PROGRAM DNS_DYN_DEMO
VAR
	DNS_DYN : DNS_DYN;
	IP_C : IP_C;
	S_BUF : NETWORK_BUFFER;
	R_BUF : NETWORK_BUFFER;
	IP_CONTROL : IP_CONTROL;
	enable: BOOL;
	done : BOOL;
	error_c : DWORD;
	error_t : BYTE;
	busy : BOOL;
	COUNT_DR: COUNT_DR;
	z: DWORD;

	GET_WAN_IP : GET_WAN_IP;
	t1: TON;
	done2 : BOOL;
	error_c2 : DWORD;
	error_t2 : BYTE;
	update : BOOL;
	new_ip: BOOL;
	wan_ip4: DWORD;
END_VAR
VAR // added by the converter: edge detectors and wires of the graphical bodies
    _w1 : ANY;
END_VAR

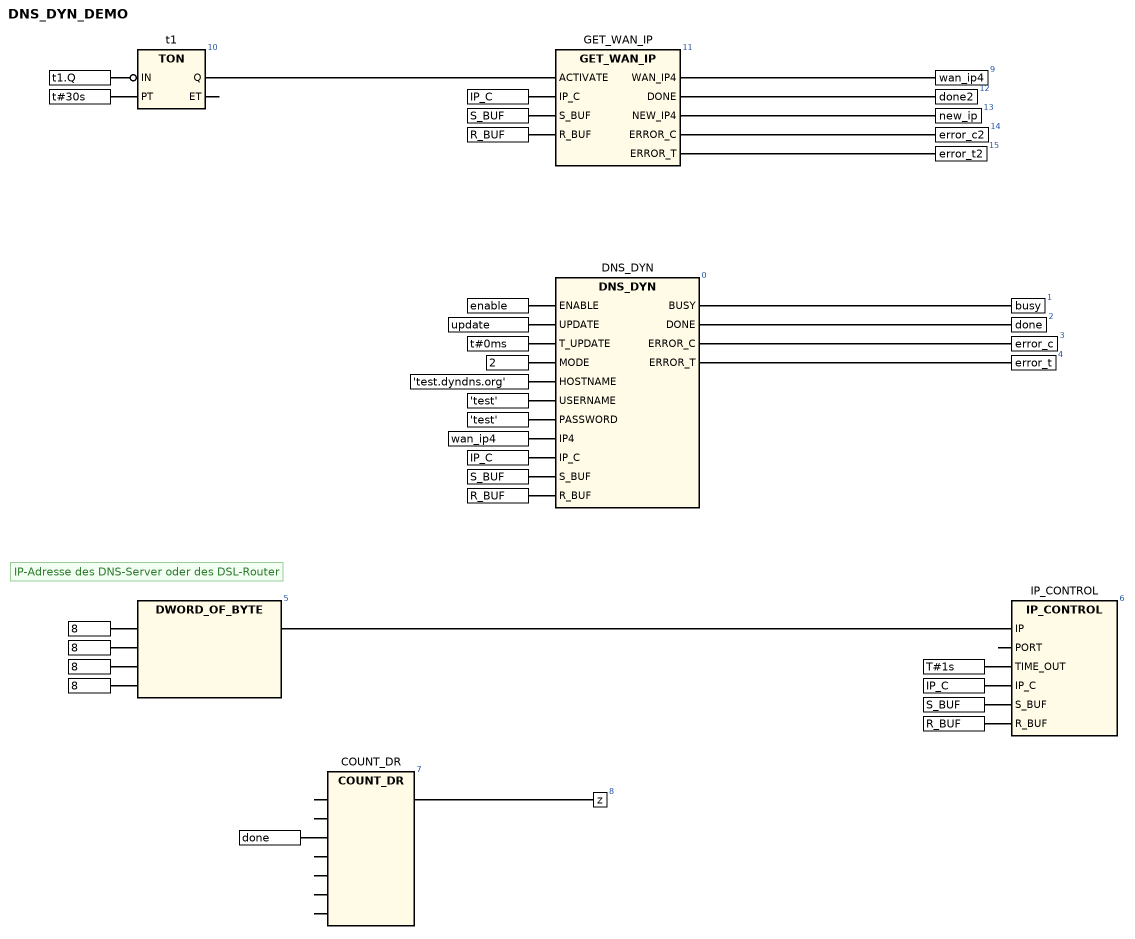
DNS_DYN(
    ENABLE := enable,
    UPDATE := update,
    T_UPDATE := t#0ms,
    MODE := 2,
    HOSTNAME := 'test.dyndns.org',
    USERNAME := 'test',
    PASSWORD := 'test',
    IP4 := wan_ip4,
    IP_C := IP_C,
    S_BUF := S_BUF,
    R_BUF := R_BUF);
busy := DNS_DYN.BUSY;
done := DNS_DYN.DONE;
error_c := DNS_DYN.ERROR_C;
error_t := DNS_DYN.ERROR_T;
// IP-Adresse des DNS-Server oder des DSL-Router
_w1 := DWORD_OF_BYTE(8, 8, 8, 8);
IP_CONTROL(IP := _w1, TIME_OUT := T#1s, IP_C := IP_C, S_BUF := S_BUF, R_BUF := R_BUF);
COUNT_DR(_in3 := done);
z := COUNT_DR._out1;
wan_ip4 := GET_WAN_IP.WAN_IP4;
t1(IN := NOT t1.Q, PT := t#30s); // TON
GET_WAN_IP(ACTIVATE := t1.Q, IP_C := IP_C, S_BUF := S_BUF, R_BUF := R_BUF);
done2 := GET_WAN_IP.DONE;
new_ip := GET_WAN_IP.NEW_IP4;
error_c2 := GET_WAN_IP.ERROR_C;
error_t2 := GET_WAN_IP.ERROR_T;

END_PROGRAM

(* stored: Version 1.1.0.1, ProductVersion 3.1.4024.9
   POU DNS_DYN_DEMO: Id {1a109249-4351-4a0a-a001-36d4b101485e}, SpecialFunc None *)
